FUNCTION_BLOCK AW_FIELDBUS_WORD_TO_SIGNAL_COMPOUND_SCALE (* Mirrors IN->OUT if Signal Valid, with compound scaling for upper and lower byte *)
  (* Standard: 61499-1; Description: Copyright (c) 2026 HR Agrartechnik GmbH This program and the accompanying materials are made available under the terms of the Eclipse Public License 2.0 which is available at https://www.eclipse.org/legal/epl-2.0/ SPDX-License-Identifier: EPL-2.0 *)
  (* Version 1.0, 2026-05-31, Franz Höpfinger, HR Agrartechnik GmbH *)
  PACKAGE logiBUS::signalprocessing::fieldbus;
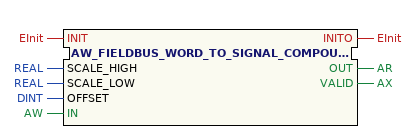
  EVENT_INPUT
    INIT : EInit; (* Init Request *)
  END_EVENT
  EVENT_OUTPUT
    INITO : EInit; (* Init Confirmation *)
  END_EVENT
  VAR_INPUT
    SCALE_HIGH : REAL := REAL#0.256; (* Scale factor for upper byte *)
    SCALE_LOW : REAL := REAL#0.001; (* Scale factor for lower byte *)
    OFFSET : DINT := DINT#0; (* Offset added after scaling *)
  END_VAR
  SOCKETS
    IN : adapter::types::unidirectional::AW; (* Input *)
  END_SOCKETS
  PLUGS
    OUT : adapter::types::unidirectional::AR; (* Output Filtered *)
    VALID : adapter::types::unidirectional::AX; (* TRUE if Signal is VALID *)
  END_PLUGS
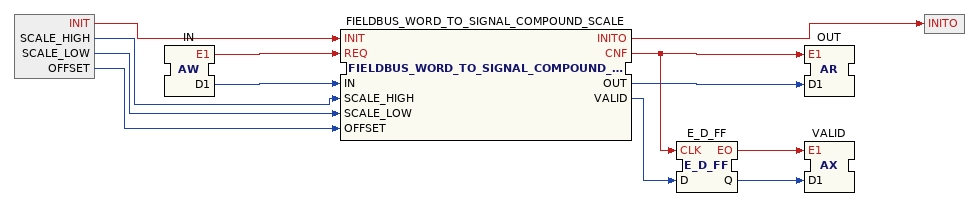
  FBS
    FIELDBUS_WORD_TO_SIGNAL_COMPOUND_SCALE : logiBUS::signalprocessing::fieldbus::FIELDBUS_WORD_TO_SIGNAL_COMPOUND_SCALE;
    E_D_FF : iec61499::events::E_D_FF;
  END_FBS
  EVENT_CONNECTIONS
    IN.E1 TO FIELDBUS_WORD_TO_SIGNAL_COMPOUND_SCALE.REQ;
    FIELDBUS_WORD_TO_SIGNAL_COMPOUND_SCALE.CNF TO OUT.E1;
    FIELDBUS_WORD_TO_SIGNAL_COMPOUND_SCALE.CNF TO E_D_FF.CLK;
    E_D_FF.EO TO VALID.E1;
    INIT TO FIELDBUS_WORD_TO_SIGNAL_COMPOUND_SCALE.INIT;
    FIELDBUS_WORD_TO_SIGNAL_COMPOUND_SCALE.INITO TO INITO;
  END_CONNECTIONS
  DATA_CONNECTIONS
    IN.D1 TO FIELDBUS_WORD_TO_SIGNAL_COMPOUND_SCALE.IN;
    FIELDBUS_WORD_TO_SIGNAL_COMPOUND_SCALE.OUT TO OUT.D1;
    FIELDBUS_WORD_TO_SIGNAL_COMPOUND_SCALE.VALID TO E_D_FF.D;
    E_D_FF.Q TO VALID.D1;
    SCALE_HIGH TO FIELDBUS_WORD_TO_SIGNAL_COMPOUND_SCALE.SCALE_HIGH;
    SCALE_LOW TO FIELDBUS_WORD_TO_SIGNAL_COMPOUND_SCALE.SCALE_LOW;
    OFFSET TO FIELDBUS_WORD_TO_SIGNAL_COMPOUND_SCALE.OFFSET;
  END_CONNECTIONS
END_FUNCTION_BLOCK
